Staubli VAL3: Form_Welcome.pgx

public program Form_Welcome(string x_sTitle, bool& x_bExit)
begin
  //欢迎界面，显示日期和时间
  userPage()
  cls()
  title(x_sTitle)
  call Control_PanelMd("欢迎使用史陶比尔机器人软件")

  while !x_bExit
    gotoxy(1,12)
    put(left("时间:"+getDate("%H:%M:%S"),30))
    gotoxy(1,13)
    put(left("日期:"+getDate("%Y")+"年"+getDate("%m")+"月"+getDate("%d")+"日",30))
    delay(0)
  endWhile



end
